// TwinCAT 3 PLC project Main
// ProgramVersion: 3.1.4026.21
// libraries:
//   Tc2_MC2, * (Beckhoff Automation GmbH)
//   Tc2_Standard, * (Beckhoff Automation GmbH)
//   Tc2_System, * (Beckhoff Automation GmbH)
// project tree:
//   / PlcTask.TcTTO
//   POUs/ MAIN.TcPOU, NUMBA.TcDUT, TESTE.TcDUT, TestStruct.TcDUT

CONFIGURATION Main
    RESOURCE PLC ON TwinCAT3
        TASK PlcTask(INTERVAL := T#10ms, PRIORITY := 20);
        PROGRAM MAIN WITH PlcTask : MAIN;
    END_RESOURCE
END_CONFIGURATION

// ---- POUs/NUMBA.TcDUT
TYPE NUMBA :
STRUCT
	More: LREAL;
	Dizasta: TESTE;
	bleeks: DWORD;
	moar: TestStruct;
END_STRUCT
END_TYPE

// ---- POUs/TESTE.TcDUT
{attribute 'qualified_only'}
{attribute 'strict'}
{attribute 'to_string'}
TYPE TESTE :
(
	enum_member := 0,
	blarhg
);
END_TYPE

// ---- POUs/TestStruct.TcDUT
TYPE TestStruct :
STRUCT
	i: INT;
	b: REAL;
	test_array_st: ARRAY[0..12] OF LREAL;
END_STRUCT
END_TYPE

// ---- POUs/MAIN.TcPOU
PROGRAM MAIN
VAR
	i : INT;
	b: REAL;
	change_int: INT;
	state: UINT;
	start: BOOL;
	eeks: TestStruct;
	beeks: TestStruct;
	theetest: TESTE;
	today: DATE;
	timetest: TIME := T#25S;
	dt_test : DT;
	masta_disasta: NUMBA;
	test_array: ARRAY[0..12] OF INT;
	blargh: TOD;
	ArrayOfStructs: ARRAY[1..5] OF NUMBA;
	dastring : STRING := 'BOB';
	longint: LINT := 300;
	lwordtest: LWORD := 12435;
	ulintdsaaa: ULINT := 214321;
END_VAR

i := i + 1;
eeks.b := i *2;

END_PROGRAM
